// TIA Portal V20 export
DATA_BLOCK "BK16"   // DB300
// stored: MemoryReserve 100
   VAR
      "X10-1.CATHODE NG P&P 1st BACKWARD" : Bool := TRUE;
      "X11-1.SPARE" : Bool := FALSE;
      "X12-1.CATHODE NG P&P 2nd BACKWARD" : Bool := TRUE;
      "X13-1.SPARE" : Bool := FALSE;
      "X14-1.CATHODE NG P&P DOWN" : Bool := TRUE;
      "X15-1.SPARE" : Bool := FALSE;
      "X16-1.CATHODE NG P&P VACUUM PRESSURE SWITCH" : Bool := FALSE;
      "X17-1.SPARE" : Bool := FALSE;
      "X10-2.CATHODE NG P&P 1st FORWARD" : Bool := FALSE;
      "X11-2.SPARE" : Bool := FALSE;
      "X12-2.CATHODE NG P&P 2nd FORWARD" : Bool := FALSE;
      "X13-2.SPARE" : Bool := FALSE;
      "X14-2.CATHODE NG P&P UP" : Bool := FALSE;
      "X15-2.SPARE" : Bool := FALSE;
      "X16-2.CATHODE NG P&P ELECTRODE DETECT SENSOR" : Bool := FALSE;
      "X17-2.SPARE" : Bool := FALSE;
   END_VAR
BEGIN
END_DATA_BLOCK
